Universal Robots PolyScope program: visionsimple.urp

Program visionsimple (installation=default directory=/home/ur/ursim-current/programs createdIn=3.2.18654.0 lastSavedIn=5.11.9.1010452 robotSerialNumber=20195599999)
Calibrated DH parameters: a=[0, -0.425, -0.3922, 0, 0, 0]; d=[0.1625, 0, 0, 0.1333, 0.0997, 0.0996]; alpha=[1.570796, 0, 0, 1.570796, -1.570796, 0]; deltaTheta=[0, 0, 0, 0, 0, 0]
Robot Program (runOnlyOnce=false)
  MoveJ speed 60 deg/s, acceleration 80 deg/s^2 (useActiveTCP=false) feature=Base
    Waypoint punto_ref: TCP in base x=-115.755 y=-608.104 z=633.047 mm, rx=-0.0288 ry=2.2249 rz=-2.1435 rad; joints [-88.584, -105.185, -80.022, 3.108, 91.471, 1.353] deg
  Folder Datos_Recibidos_Camara
    'Esperar la foto realizada por la camara'
    x := 400
    y := 200
    rz := 30
  Folder Calcular_Posicion_Pick
    '# Convert mm to m and deg to rad'
    pos_base_camara := p[(x/1000), (y/1000), 0, 0, 0, d2r(rz)]
    pos_pick := pose_trans(punto_ref, pos_base_camara)
  Folder Mover_a_pos_pick
    MoveL speed 250 mm/s, acceleration 1200 mm/s^2 (useActiveTCP=true) feature=Base
      Waypoint Waypoint (Variable): variable=pos_pick
